// SIMATIC STEP 7 (V5.x) project 315客户机
// CPU: CPU315-2 PN/DP(1)
// station: P_ADR_BUS
// station: 硬件
// station: SIMATIC 300 站点
// program: S7 程序(1)

SYMBOL_TABLE
"Cycle Execution"	OB 1	OB 1
"CYC_INT5"	OB 35	OB 35	// Cyclic Interrupt 5
"I/O_FLT1"	OB 82	OB 82	// I/O Point Fault 1
"OBNL_FLT"	OB 85	OB 85	// OB Not Loaded Fault
"RACK_FLT"	OB 86	OB 86	// Loss of Rack Fault
"COMPLETE RESTART"	OB 100	OB 100	// Complete Restart
"MOD_ERR"	OB 122	OB 122	// Module Access Error
"GET"	SFB 14	SFB 14	// Read Data From a Remote CPU
"PUT"	SFB 15	SFB 15	// Write Data to a Remote CPU
"FILL"	SFC 21	SFC 21	// Initialize a Memory Area
"VAT_1"	VAT 1	
END_SYMBOL_TABLE

// FB 14: know-how protected block, not included

// FB 15: know-how protected block, not included

DATA_BLOCK DB 1
VERSION : 0.1
  STRUCT
   ARAY : ARRAY  [0 .. 200 ] OF BYTE ;
  END_STRUCT ;	
BEGIN
END_DATA_BLOCK

DATA_BLOCK DB 2
VERSION : 0.1
  STRUCT
   ARAY : ARRAY  [0 .. 200 ] OF BYTE ;
  END_STRUCT ;	
BEGIN
END_DATA_BLOCK

DATA_BLOCK DB 14
AUTHOR : SIMATIC
FAMILY : CPU_300
VERSION : 0.0
FB 14
BEGIN
END_DATA_BLOCK

DATA_BLOCK DB 15
AUTHOR : SIMATIC
FAMILY : CPU_300
VERSION : 0.0
FB 15
BEGIN
END_DATA_BLOCK

ORGANIZATION_BLOCK "Cycle Execution"	// OB 1
TITLE = "Main Program Sweep (Cycle)"
VERSION : 0.1
VAR_TEMP
  OB1_EV_CLASS : BYTE ;	//Bits 0-3 = 1 (Coming event), Bits 4-7 = 1 (Event class 1)
  OB1_SCAN_1 : BYTE ;	//1 (Cold restart scan 1 of OB 1), 3 (Scan 2-n of OB 1)
  OB1_PRIORITY : BYTE ;	//Priority of OB Execution
  OB1_OB_NUMBR : BYTE ;	//1 (Organization block 1, OB1)
  OB1_RESERVED_1 : BYTE ;	//Reserved for system
  OB1_RESERVED_2 : BYTE ;	//Reserved for system
  OB1_PREV_CYCLE : INT ;	//Cycle time of previous OB1 scan (milliseconds)
  OB1_MIN_CYCLE : INT ;	//Minimum cycle time of OB1 (milliseconds)
  OB1_MAX_CYCLE : INT ;	//Maximum cycle time of OB1 (milliseconds)
  OB1_DATE_TIME : DATE_AND_TIME ;	//Date and time OB1 started
END_VAR
BEGIN
NETWORK
TITLE = 时钟脉冲信号反相
      AN    M 8.1;
      =     M 10.0;
NETWORK
TITLE = 读取通信伙伴的数据
      CALL  FB 14 , DB 14 (
           DIX 0.0                  := M 8.1,
           DIW 2                    := 1,
           DIX 4.0                  := M 0.1,
           DIX 4.1                  := M 0.2,
           DIW 6                    := MW 2,
           DIW 8                    := W#16#1002,
           DIW 10                   := 200,
           DIW 12                   := 1,
           DID 14                   := P#DBX 100.0,
           DIW 18                   := W#16#1002,
           DIW 20                   := 200,
           DIW 22                   := 2,
           DID 24                   := P#DBX 0.0);	//ÉÏÉýÑØÊ±¼¤»îÊý¾Ý´«Êä£¬Ã¿200ms¶ÁÈ¡Ò»´Î / S7Á¬½ÓºÅ / Ã¿´Î¶ÁÈ¡Íê³É²úÉúÒ»¸öÂö³å / ´íÎó±êÖ¾£¬³ö´íÊ±Îª1 / ×´Ì¬×Ö£¬Îª0Ê±±íÊ¾Ã»ÓÐ¾¯¸æºÍ´íÎó / Òª¶ÁÈ¡µÄS7-200 SMARTµÄVB100¡«VB299 / ±¾Õ¾´æ·Å¶ÁÈ¡µÄÊý¾ÝµÄµØÖ·Çø
NETWORK
TITLE = 向通信伙伴的数据区写入数据
      CALL  FB 15 , DB 15 (
           DIX 0.0                  := M 10.0,
           DIW 2                    := 1,
           DIX 4.0                  := M 10.1,
           DIX 4.1                  := M 10.2,
           DIW 6                    := MW 12,
           DIW 8                    := W#16#1002,
           DIW 10                   := 200,
           DIW 12                   := 1,
           DID 14                   := P#DBX 300.0,
           DIW 18                   := W#16#1002,
           DIW 20                   := 200,
           DIW 22                   := 1,
           DID 24                   := P#DBX 0.0);	//ÉÏÉýÑØÊ±¼¤»îÊý¾Ý½»»»£¬Ã¿200msÐ´Ò»´Î / S7Á¬½ÓºÅ / Ã¿´ÎÐ´²Ù×÷Íê³É²úÉúÒ»¸öÂö³å / ´íÎó±êÖ¾£¬³ö´íÊ±Îª1 / ×´Ì¬×Ö£¬Îª0Ê±±íÊ¾Ã»ÓÐ¾¯¸æºÍ´íÎó / ÒªÐ´ÈëÊý¾ÝµÄS7-200 SMARTµÄVB300¡«VB499 / ´æ·Å±¾Õ¾Òª·¢ËÍµÄÊý¾ÝµÄµØÖ·Çø
END_ORGANIZATION_BLOCK

ORGANIZATION_BLOCK "CYC_INT5"	// OB 35
TITLE = "Cyclic Interrupt"
VERSION : 0.1
VAR_TEMP
  OB35_EV_CLASS : BYTE ;	//Bits 0-3 = 1 (Coming event), Bits 4-7 = 1 (Event class 1)
  OB35_STRT_INF : BYTE ;	//16#36 (OB 35 has started)
  OB35_PRIORITY : BYTE ;	//Priority of OB Execution
  OB35_OB_NUMBR : BYTE ;	//35 (Organization block 35, OB35)
  OB35_RESERVED_1 : BYTE ;	//Reserved for system
  OB35_RESERVED_2 : BYTE ;	//Reserved for system
  OB35_PHASE_OFFSET : WORD ;	//Phase offset (msec)
  OB35_RESERVED_3 : INT ;	//Reserved for system
  OB35_EXC_FREQ : INT ;	//Frequency of execution (msec)
  OB35_DATE_TIME : DATE_AND_TIME ;	//Date and time OB35 started
END_VAR
BEGIN
NETWORK
TITLE =
      L     DB1.DBW 0;
      +     1;
      T     DB1.DBW 0;
END_ORGANIZATION_BLOCK

ORGANIZATION_BLOCK "I/O_FLT1"	// OB 82
TITLE = "I/O Point Fault"
VERSION : 0.1
VAR_TEMP
  OB82_EV_CLASS : BYTE ;	//16#39, Event class 3, Entering event state, Internal fault event
  OB82_FLT_ID : BYTE ;	//16#XX, Fault identifcation code
  OB82_PRIORITY : BYTE ;	//Priority of OB Execution
  OB82_OB_NUMBR : BYTE ;	//82 (Organization block 82, OB82)
  OB82_RESERVED_1 : BYTE ;	//Reserved for system
  OB82_IO_FLAG : BYTE ;	//Input (01010100), Output (01010101)
  OB82_MDL_ADDR : WORD ;	//Base address of module with fault
  OB82_MDL_DEFECT : BOOL ;	//Module defective
  OB82_INT_FAULT : BOOL ;	//Internal fault
  OB82_EXT_FAULT : BOOL ;	//External fault
  OB82_PNT_INFO : BOOL ;	//Point information
  OB82_EXT_VOLTAGE : BOOL ;	//External voltage low
  OB82_FLD_CONNCTR : BOOL ;	//Field wiring connector missing
  OB82_NO_CONFIG : BOOL ;	//Module has no configuration data
  OB82_CONFIG_ERR : BOOL ;	//Module has configuration error
  OB82_MDL_TYPE : BYTE ;	//Type of module
  OB82_SUB_MDL_ERR : BOOL ;	//Sub-Module is missing or has error
  OB82_COMM_FAULT : BOOL ;	//Communication fault
  OB82_MDL_STOP : BOOL ;	//Module is stopped
  OB82_WTCH_DOG_FLT : BOOL ;	//Watch dog timer stopped module
  OB82_INT_PS_FLT : BOOL ;	//Internal power supply fault
  OB82_PRIM_BATT_FLT : BOOL ;	//Primary battery is in fault
  OB82_BCKUP_BATT_FLT : BOOL ;	//Backup battery is in fault
  OB82_RESERVED_2 : BOOL ;	//Reserved for system
  OB82_RACK_FLT : BOOL ;	//Rack fault, only for bus interface module
  OB82_PROC_FLT : BOOL ;	//Processor fault
  OB82_EPROM_FLT : BOOL ;	//EPROM fault
  OB82_RAM_FLT : BOOL ;	//RAM fault
  OB82_ADU_FLT : BOOL ;	//ADU fault
  OB82_FUSE_FLT : BOOL ;	//Fuse fault
  OB82_HW_INTR_FLT : BOOL ;	//Hardware interupt input in fault
  OB82_RESERVED_3 : BOOL ;	//Reserved for system
  OB82_DATE_TIME : DATE_AND_TIME ;	//Date and time OB82 started
END_VAR
BEGIN
// (block stored without names or comments; labels and parameter names are numbered)
END_ORGANIZATION_BLOCK

ORGANIZATION_BLOCK "RACK_FLT"	// OB 86
TITLE = "Loss Of Rack Fault"
VERSION : 0.1
VAR_TEMP
  OB86_EV_CLASS : BYTE ;	//16#38/39 Event class 3
  OB86_FLT_ID : BYTE ;	//16#C1/C4/C5, Fault identifcation code
  OB86_PRIORITY : BYTE ;	//Priority of OB Execution
  OB86_OB_NUMBR : BYTE ;	//86 (Organization block 86, OB86)
  OB86_RESERVED_1 : BYTE ;	//Reserved for system
  OB86_RESERVED_2 : BYTE ;	//Reserved for system
  OB86_MDL_ADDR : WORD ;	//Base address of IM module in rack with fault
  OB86_RACKS_FLTD : ARRAY  [0 .. 31 ] OF BOOL ;	//Racks in fault
  OB86_DATE_TIME : DATE_AND_TIME ;	//Date and time OB86 started
END_VAR
BEGIN
// (block stored without names or comments; labels and parameter names are numbered)
END_ORGANIZATION_BLOCK

ORGANIZATION_BLOCK "COMPLETE RESTART"	// OB 100
TITLE = "Complete Restart"
VERSION : 0.1
VAR_TEMP
  OB100_EV_CLASS : BYTE ;	//16#13, Event class 1, Entering event state, Event logged in diagnostic buffer
  OB100_STRTUP : BYTE ;	//16#81/82/83/84 Method of startup
  OB100_PRIORITY : BYTE ;	//Priority of OB Execution
  OB100_OB_NUMBR : BYTE ;	//100 (Organization block 100, OB100)
  OB100_RESERVED_1 : BYTE ;	//Reserved for system
  OB100_RESERVED_2 : BYTE ;	//Reserved for system
  OB100_STOP : WORD ;	//Event that caused CPU to stop (16#4xxx)
  OB100_STRT_INFO : DWORD ;	//Information on how system started
  OB100_DATE_TIME : DATE_AND_TIME ;	//Date and time OB100 started
END_VAR
BEGIN
NETWORK
TITLE = 初始化发送数据区
      L     W#16#4001;
      T     LW 20;
      CALL  "FILL" (
           BVAL                     := P#L 20.0 WORD 1,
           RET_VAL                  := LW 22,
           BLK                      := P#DB1.DBX 0.0 BYTE 20);	//Ô´Êý¾Ý / ¹ÊÕÏ´úÂë / µØÖ·Çø
NETWORK
TITLE = 接收数据区清零
      L     W#16#0;
      T     LW 20;
      CALL  "FILL" (
           BVAL                     := P#L 20.0 WORD 1,
           RET_VAL                  := LW 22,
           BLK                      := P#DB2.DBX 0.0 BYTE 20);	//Ô´Êý¾Ý / ¹ÊÕÏ´úÂë / µØÖ·Çø
END_ORGANIZATION_BLOCK

ORGANIZATION_BLOCK "MOD_ERR"	// OB 122
TITLE = "Module Access Error"
VERSION : 0.1
VAR_TEMP
  OB122_EV_CLASS : BYTE ;	//16#25, Event class 2, Entering event state, Internal fault event
  OB122_SW_FLT : BYTE ;	//16#XX Software error code
  OB122_PRIORITY : BYTE ;	//Priority of OB Execution
  OB122_OB_NUMBR : BYTE ;	//122 (Organization block 122, OB122)
  OB122_BLK_TYPE : BYTE ;	//16#88/8A/8B/8C/8E Type of block fault occured in
  OB122_MEM_AREA : BYTE ;	//Memory area where access error occured
  OB122_MEM_ADDR : WORD ;	//Memory address where access error occured
  OB122_BLK_NUM : WORD ;	//Block number in which error occured
  OB122_PRG_ADDR : WORD ;	//Program address where error occured
  OB122_DATE_TIME : DATE_AND_TIME ;	//Date and time OB1 started
END_VAR
BEGIN
// (block stored without names or comments; labels and parameter names are numbered)
END_ORGANIZATION_BLOCK
